// SIMATIC S7-200 SMART project (STEP 7-Micro/WIN SMART), CPU SR40

SYMBOL_TABLE 系统符号
Always_On        SM0.0    // 始终接通
First_Scan_On    SM0.1    // 仅在第一个扫描周期时接通
Clock_1s         SM0.5    // 针对 1 s 的周期时间，时钟脉冲接通 0.5 s，断开 0.5 s.
END_SYMBOL_TABLE

ORGANIZATION_BLOCK MAIN:OB1
TITLE=程序注释
BEGIN
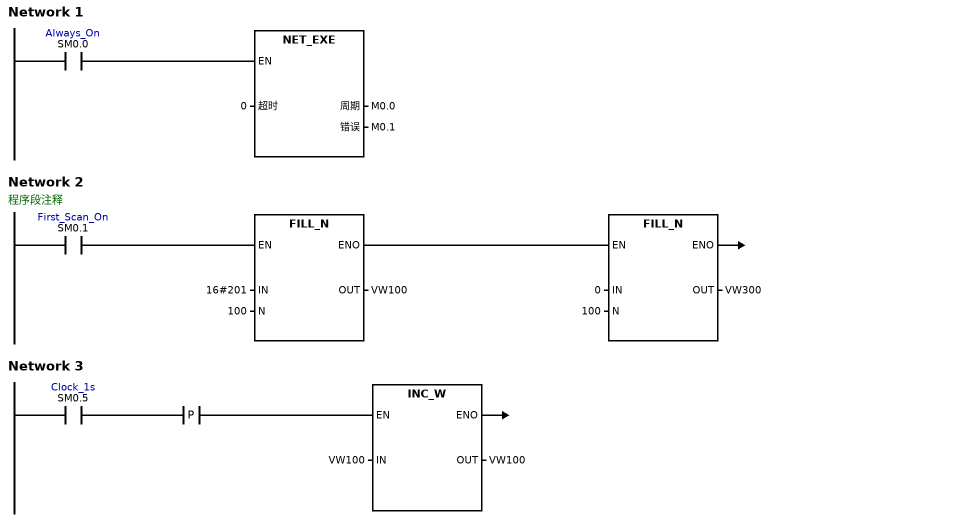
Network 1
LD     Always_On:SM0.0
CALL   NET_EXE:SBR1, 0, M0.0, M0.1
Network 2
// 程序段注释
// (network saved uncompiled; LAD cells follow)
// row 0: c0 -| |- First_Scan_On:SM0.1  c1 --  c2 [FILL_N EN:=power@row0, IN:=16#201, N:=100, ENO=>power, OUT=>VW100]  c3 --  c4 --  c5 [FILL_N EN:=power@row0, IN:=0, N:=100, ENO=>power, OUT=>VW300]  c6 ->
// row 1: c2 [box]  c5 [box]
Network 3
LD     Clock_1s:SM0.5
EU
INCW   VW100
END_ORGANIZATION_BLOCK

// SBR1: protected block, not included
